// Mitsubishi GX Works2 project: z08   PLC: Q02/Q02H

PROGRAM MAIN
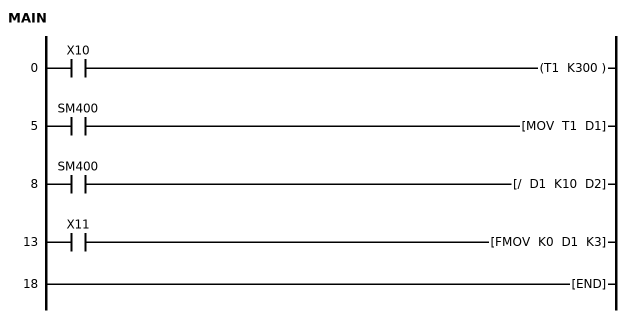
0     LD      X10
      OUT     T1 K300
5     LD      SM400
      MOV     T1 D1
8     LD      SM400
      /       D1 K10 D2
13    LD      X11
      FMOV    K0 D1 K3
18    END
END_PROGRAM
